// Mitsubishi GX Works2 project: LRI.gx3   PLC: Q03UDV
// V1

PROGRAM MAIN
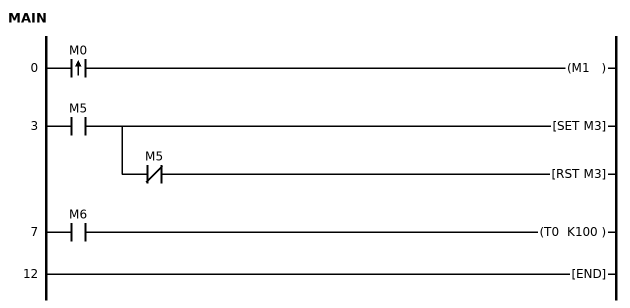
0     LDP     M0
      OUT     M1
3     LD      M5
      SET     M3
      ANI     M5
      RST     M3
7     LD      M6
      OUT     T0 K100
12    END
END_PROGRAM
